// TIA Portal project "stl_demo_1" (V15)

(* hardware
DEVICE "S7-1200 station_1"  S7-1200 Station
   slot 0: "Rack_0"  S7-1200 Rack  Rack  V1.0
   slot 1: "PLC_1"  CPU 1214C DC/DC/DC  6ES7 214-1AG40-0XB0  V4.2
*)

// ===== PLC "PLC_1"  CPU 1214C DC/DC/DC =====

VAR_GLOBAL   // PLC tag table "Default tag table"
   "DIAMETER" AT %IW0 : Int;
   "OUT_01" AT %M4.0 : Bool;
   "TRIG_F1" AT %M100.0 : Bool;
   "Tag_1" AT %M200.0 : Bool;
   "TRIG_F2" AT %M100.1 : Bool;
END_VAR

FUNCTION "Block_1" : Void   // FC1, LAD
{ S7_Optimized_Access := 'TRUE' }
VERSION : 0.1
   VAR_INPUT
      DIAMETER : Int;
   END_VAR
   VAR_OUTPUT
      OUTPUT_1 : Bool;
   END_VAR
BEGIN

REGION Network 1 (SCL)
   IF #DIAMETER >0 THEN
       #OUTPUT_1 := TRUE;
   ELSE
       #OUTPUT_1 := FALSE;
   END_IF;
END_REGION
END_FUNCTION

ORGANIZATION_BLOCK "Main"   // OB1, LAD, ProgramCycle
TITLE = "Main Program Sweep (Cycle)"
{ S7_Optimized_Access := 'TRUE' }
VERSION : 0.1
   VAR_INPUT
      Initial_Call : Bool;   // Initial call of this OB
      Remanence : Bool;   // =True, if remanent data are available
   END_VAR
BEGIN

REGION Network 1
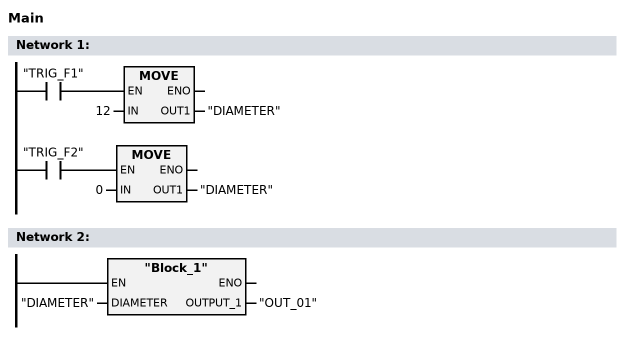
   RUNG wire#powerrail
      Contact( "TRIG_F1" )
      Move(in := 12, out1 => "DIAMETER")
   END_RUNG
   RUNG wire#powerrail
      Contact( "TRIG_F2" )
      Move(in := 0, out1 => "DIAMETER")
   END_RUNG
   // the same network as SCL:
   IF "TRIG_F1" THEN "DIAMETER" := 12; END_IF;
   IF "TRIG_F2" THEN "DIAMETER" := 0; END_IF;
END_REGION

REGION Network 2
   RUNG wire#powerrail
      "Block_1"(DIAMETER := "DIAMETER", OUTPUT_1 => "OUT_01")
   END_RUNG
   // the same network as SCL:
   "Block_1"(DIAMETER := "DIAMETER", OUTPUT_1 => "OUT_01");
END_REGION
END_ORGANIZATION_BLOCK